(* PLC project  *)

CONFIGURATION Application
  RESOURCE Application ON PLC
    TASK BusTask(INTERVAL := T#4ms, PRIORITY := 1);
    PROGRAM app WITH BusTask : app;
  END_RESOURCE
END_CONFIGURATION
